{attribute 'GeneratedUsingTerminal: EPP2816-0008-0016'}
{attribute addProperty BoxType "EPP2816-0008-0016"}
{attribute addProperty Id "EtcSlaveTerminalBaseDIG_Diag_Inputs_Channel_1AT %I*DIG_Diag_Inputs_Channel_584303BF8DIG_Diag_Inputs_Channel_2AT %I*DIG_Diag_Inputs_Channel_584303BF8DIG_Inputs_DeviceAT %I*DIG_Inputs_Device_E94E5BF95DIG_Outputs_Channel_1AT %Q*DIG_Outputs_Channel_28AC1A9E8DIG_Outputs_Channel_2AT %Q*DIG_Outputs_Channel_28AC1A9E8DIG_Outputs_DeviceAT %Q*DIG_Outputs_Device_36A5EF172WcStateAT %I*WcState_9091E0EB2InfoDataAT %I*InfoData_32EB74EA10"}
{attribute addProperty CRC "775918764"}
{attribute addProperty Size "51"}
TYPE EPP2816_2E3F94AC EXTENDS EtcSlaveTerminalBase :
STRUCT
	{attribute addProperty Name "DIG_Diag_Inputs_Channel_1"}
	DIG_Diag_Inputs_Channel_1 : DIG_Diag_Inputs_Channel_584303BF;
	{attribute addProperty Name "DIG_Diag_Inputs_Channel_2"}
	DIG_Diag_Inputs_Channel_2 : DIG_Diag_Inputs_Channel_584303BF;
	{attribute addProperty Name "DIG_Inputs_Device"}
	DIG_Inputs_Device : DIG_Inputs_Device_E94E5BF9;
	{attribute addProperty Name "DIG_Outputs_Channel_1"}
	DIG_Outputs_Channel_1 : DIG_Outputs_Channel_28AC1A9E;
	{attribute addProperty Name "DIG_Outputs_Channel_2"}
	DIG_Outputs_Channel_2 : DIG_Outputs_Channel_28AC1A9E;
	{attribute addProperty Name "DIG_Outputs_Device"}
	DIG_Outputs_Device : DIG_Outputs_Device_36A5EF17;
	{attribute addProperty Name "WcState"}
	WcState : WcState_9091E0EB;
	{attribute addProperty Name "InfoData"}
	InfoData : InfoData_32EB74EA;
END_STRUCT
END_TYPE

(* stored: Version 1.2.0.0, ProductVersion 3.1.4024.9
   DUT EPP2816_2E3F94AC: Id {73cdff1b-4ad5-41a0-811a-a01f172be986} *)
